// TIA Portal V20 export
// export: Created 2026-10-03T18:54:34.8443728Z, ExportSetting WithDefaults, DisplayName Totally Integrated Automation Portal, DisplayVersion V20 Update 4, DisplayName TIA Portal Openness, DisplayVersion V20 Update 4, DisplayName TIA Portal Version Control Interface, DisplayVersion V20 Update 4, DisplayName SINAMICS Startdrive Advanced, DisplayVersion V20 SP1 Update 1, DisplayName SINAMICS Startdrive G110M, G120, G120C, G120D, G120P, G115D, DisplayVersion V20 SP1 Update 1, DisplayName SINAMICS Startdrive G130, G150, S120, S150, SINAMICS MV, G220, S200, S210, DisplayVersion V20 SP1 Update 1, DisplayName STEP 7 Professional, DisplayVersion V20 Update 4, DisplayName STEP 7 Safety, DisplayVersion V20 Update 2, DisplayName WinCC Basic/Comfort/Advanced, DisplayVersion V20 Update 4, DisplayName WinCC Unified, DisplayVersion V20 Update 4
FUNCTION "SLC_FROM_TIME" : Int   // FC24, SCL
TITLE = TIME to SLC timer counts
{ S7_Optimized_Access := 'TRUE' }
VERSION : 0.1
// Converts a timer's PT or ET back to counts of the SLC timebase, for logic that used .PRE or .ACC as a number
//  in math or moves ("time remaining" displays and the like).
// stored: AutoNumber true, IsIECCheckEnabled false, SetENOAutomatically false, UDAEnableTagReadback false
   VAR_INPUT
      Value : Time;   // Timer preset (PT) or elapsed time (ET)
      BaseMs : DInt;   // Timebase in milliseconds: 1000 for 1.0 s, 10 for 0.01 s, 1 for 0.001 s
   END_VAR
   VAR_TEMP
      counts : DInt;
   END_VAR
BEGIN
   // Whole counts, truncated like the SLC accumulator.
   #counts := TIME_TO_DINT(#Value) / #BaseMs;

   // SLC timer words are 16-bit; keep the result in that range instead of overflowing.
   IF #counts > 32767 THEN
       #counts := 32767;
   END_IF;

   #SLC_FROM_TIME := DINT_TO_INT(#counts);
END_FUNCTION
